// TIA Portal V20 export
TYPE "LAxisCtrl_typeGearInAbsolute"
TITLE = LAxisCtrl_typeGearInAbsolute
// Support: tech.team.motioncontrol@siemens.com 
// Fax: +49 (0) 9131/98-1297
   STRUCT
      ratioNumerator : DInt := 1;   // Gear ratio numerator
      ratioDenominator : DInt := 1;   // Gear ratio denominator
      masterSyncPosition : LReal := 0.0;   // Synchronous position of leading axis
      slaveSyncPosition : LReal := 0.0;   // Synchronous position of following axis
      syncProfileReference : DInt := 1;   // Type of synchronization (0: Synchronization using dynamic parameters; 1: Synchronization using leading value distance)
      masterStartDistance : LReal := 0.0;   // Leading value distance (when "SyncProfileReference" = 1)
      velocity : LReal := -1.0;   // Velocity for synchronization (when "SyncProfileReference" = 0; Value > 0.0: The specified value is used; Value = 0.0: Not permitted; Value < 0.0: Use of the default value configured in the technology object)
      acceleration : LReal := -1.0;   // Acceleration for synchronization (when "SyncProfileReference" = 0; Value > 0.0: The specified value is used; Value = 0.0: Not permitted; Value < 0.0: Use of the default value configured in the technology object)
      deceleration : LReal := -1.0;   // Deceleration for synchronization (when "SyncProfileReference" = 0; Value > 0.0: The specified value is used; Value = 0.0: Not permitted; Value < 0.0: Use of the default value configured in the technology object)
      jerk : LReal := -1.0;   // Jerk for synchronization (when "SyncProfileReference" = 0; Value > 0.0: Smooth velocity profile, the specified value is used; Value = 0.0: Trapezoid velocity profile; Value < 0.0: Use of the default value configured in the technology object)
      syncDirection : DInt := 1;   // Direction for synchronization only in effect for axes with activated modulo setting (1: Forward direction; 2: Backward direction; 3: Shortest way)
      ratioChangeOnTheFly : Bool := FALSE;   // TRUE: Changing gear ratio on-the-fly; FALSE: Ratio change requires a new rising edge at gearInAbsolute input
   END_STRUCT;
END_TYPE
